(* POU with components common to all METS systems *)
PROGRAM C01_System
VAR
	fbCloseTCPSockets			: FB_SocketCloseAll;
	fbBasePath				: FB_SYSTEM_HardwareOS;
	//fbSystemFolders			: FB_SYSTEM_CreateFolders;
	fbCoreFolders			: FB_SYSTEM_CoreFolders;
	fbCorePaths				: FB_SYSTEM_CorePaths;
	
	fbMETSAppPath				: FB_SYSTEM_HardwareOS;
	fbMETSLogsPath				: FB_SYSTEM_HardwareOS;
	fbMETSProcessPath			: FB_SYSTEM_HardwareOS;
	
	bMETSApp_OK				: BOOL;
	bMETSLogs_OK			: BOOL;	
	bMETSProcess_OK			: BOOL;

	fbNVDataCtrl				: FB_CX_NVData_NOVRAM;
	fbSettings					: FB_CX_NVData_XMLFile;
	fbValidateSettings			: FB_SYSTEM_ValidateSettings;
	
	
	


	fbPulseNetwork			: FB_PulseGenerator;
	fbNetworkInfo				: FB_CX_NetworkInfo;
	aDisplayInfo				: ARRAY[1..6, 1..2] OF STRING(23);

	fbCloseTCPPorts			: FB_TCP_CloseAllPorts;
	fbTCPServerInitOK			: RS;

	fbDateTime				: FB_SYSTEM_DateTime;
	fbShiftMonitor				: FB_SYSTEM_ShiftMonitor;
	fbProdMonitor				: FB_SYSTEM_ProdMonitor;

	bManualChange: BOOL;
	bManualClosePorts		: BOOL;
	aNovRAMSize				: ARRAY[0..10] OF UDINT;

	fbDelayShutdown			: TON; 			(*Time to abort shutdown*)
	fbShutDown				: NT_Shutdown;
	fbAbortShutdown			: NT_AbortShutdown;
	nShutdownDelay			: DWORD;		(*Shutdown delay time*)

END_VAR
VAR // added by the converter: edge detectors and wires of the graphical bodies
    _w1 : BOOL;
END_VAR

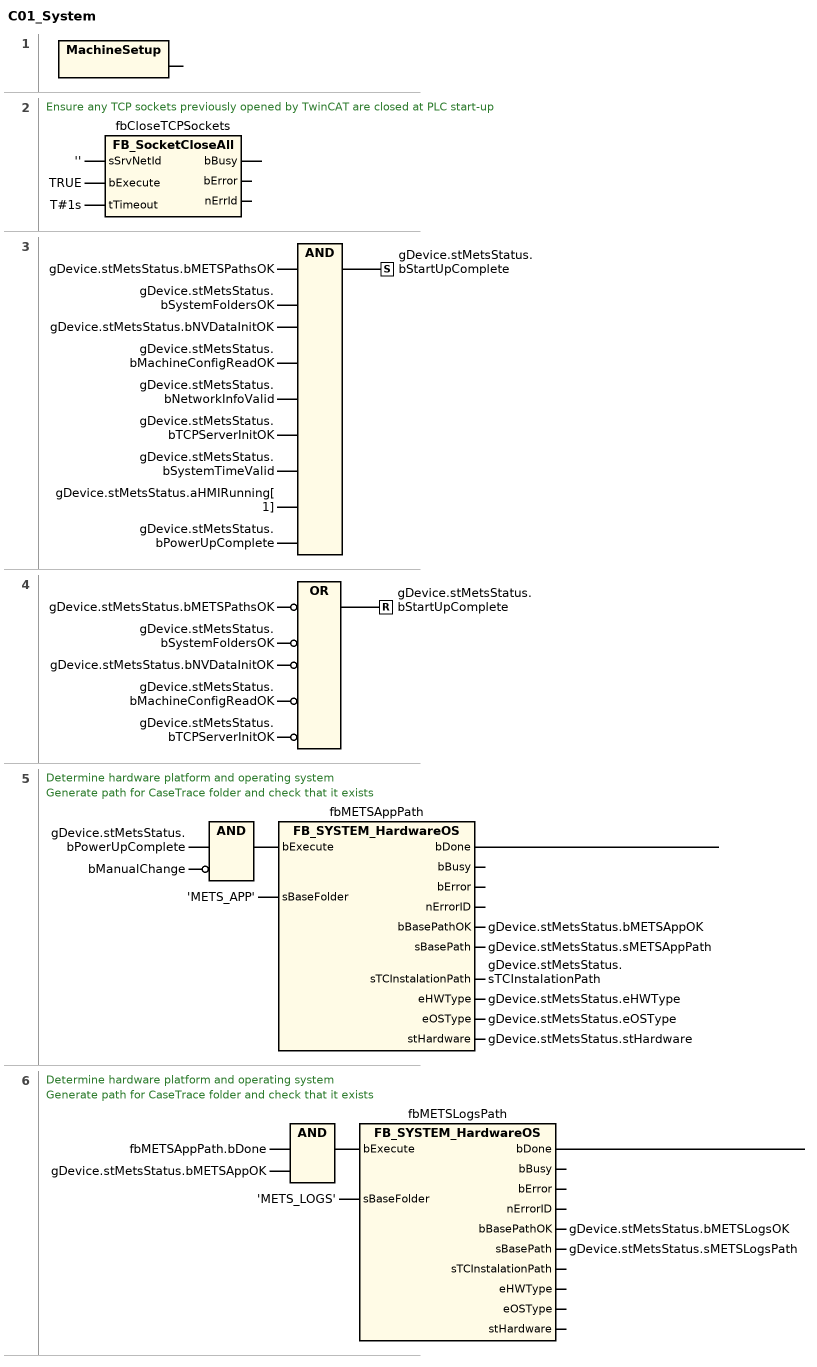
// NETWORK 1
MachineSetup();

// NETWORK 2
// Ensure any TCP sockets previously opened by TwinCAT are closed at PLC start-up
fbCloseTCPSockets(sSrvNetId := '', bExecute := TRUE, tTimeout := T#1s); // FB_SocketCloseAll

// NETWORK 3
gDevice.stMetsStatus.bStartUpComplete S= gDevice.stMetsStatus.bMETSPathsOK AND gDevice.stMetsStatus.bSystemFoldersOK AND gDevice.stMetsStatus.bNVDataInitOK AND gDevice.stMetsStatus.bMachineConfigReadOK AND gDevice.stMetsStatus.bNetworkInfoValid AND gDevice.stMetsStatus.bTCPServerInitOK AND gDevice.stMetsStatus.bSystemTimeValid AND gDevice.stMetsStatus.aHMIRunning[1] AND gDevice.stMetsStatus.bPowerUpComplete;

// NETWORK 4
gDevice.stMetsStatus.bStartUpComplete R= NOT gDevice.stMetsStatus.bMETSPathsOK OR NOT gDevice.stMetsStatus.bSystemFoldersOK OR NOT gDevice.stMetsStatus.bNVDataInitOK OR NOT gDevice.stMetsStatus.bMachineConfigReadOK OR NOT gDevice.stMetsStatus.bTCPServerInitOK;

// NETWORK 5
// 					Determine hardware platform and operating system
// Generate path for CaseTrace folder and check that it exists
//
fbMETSAppPath(
    bExecute := gDevice.stMetsStatus.bPowerUpComplete AND NOT bManualChange,
    sBaseFolder := 'METS_APP',
    bBasePathOK => gDevice.stMetsStatus.bMETSAppOK,
    sBasePath => gDevice.stMetsStatus.sMETSAppPath,
    sTCInstalationPath => gDevice.stMetsStatus.sTCInstalationPath,
    eHWType => gDevice.stMetsStatus.eHWType,
    eOSType => gDevice.stMetsStatus.eOSType,
    stHardware => gDevice.stMetsStatus.stHardware); // FB_SYSTEM_HardwareOS

// NETWORK 6
// 					Determine hardware platform and operating system
// Generate path for CaseTrace folder and check that it exists
//
fbMETSLogsPath(
    bExecute := fbMETSAppPath.bDone AND gDevice.stMetsStatus.bMETSAppOK,
    sBaseFolder := 'METS_LOGS',
    bBasePathOK => gDevice.stMetsStatus.bMETSLogsOK,
    sBasePath => gDevice.stMetsStatus.sMETSLogsPath); // FB_SYSTEM_HardwareOS

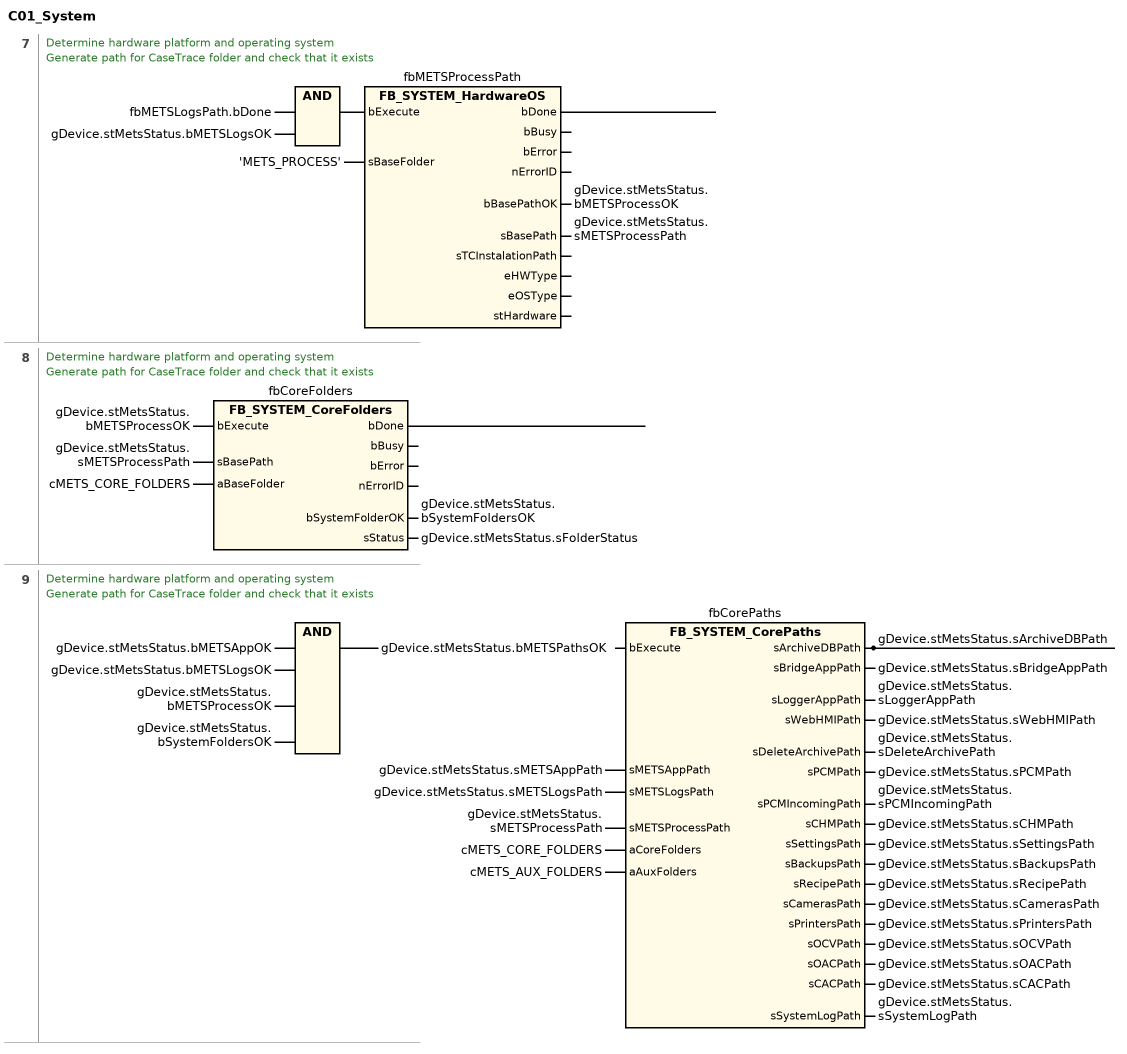
// NETWORK 7
// 					Determine hardware platform and operating system
// Generate path for CaseTrace folder and check that it exists
//
fbMETSProcessPath(
    bExecute := fbMETSLogsPath.bDone AND gDevice.stMetsStatus.bMETSLogsOK,
    sBaseFolder := 'METS_PROCESS',
    bBasePathOK => gDevice.stMetsStatus.bMETSProcessOK,
    sBasePath => gDevice.stMetsStatus.sMETSProcessPath); // FB_SYSTEM_HardwareOS

// NETWORK 8
// 					Determine hardware platform and operating system
// Generate path for CaseTrace folder and check that it exists
//
fbCoreFolders(
    bExecute := gDevice.stMetsStatus.bMETSProcessOK,
    sBasePath := gDevice.stMetsStatus.sMETSProcessPath,
    aBaseFolder := cMETS_CORE_FOLDERS,
    bSystemFolderOK => gDevice.stMetsStatus.bSystemFoldersOK,
    sStatus => gDevice.stMetsStatus.sFolderStatus); // FB_SYSTEM_CoreFolders

// NETWORK 9
// 					Determine hardware platform and operating system
// Generate path for CaseTrace folder and check that it exists
//
_w1 := gDevice.stMetsStatus.bMETSAppOK AND gDevice.stMetsStatus.bMETSLogsOK AND gDevice.stMetsStatus.bMETSProcessOK AND gDevice.stMetsStatus.bSystemFoldersOK;
gDevice.stMetsStatus.bMETSPathsOK := _w1;
fbCorePaths(
    bExecute := _w1,
    sMETSAppPath := gDevice.stMetsStatus.sMETSAppPath,
    sMETSLogsPath := gDevice.stMetsStatus.sMETSLogsPath,
    sMETSProcessPath := gDevice.stMetsStatus.sMETSProcessPath,
    aCoreFolders := cMETS_CORE_FOLDERS,
    aAuxFolders := cMETS_AUX_FOLDERS,
    sArchiveDBPath => gDevice.stMetsStatus.sArchiveDBPath,
    sBridgeAppPath => gDevice.stMetsStatus.sBridgeAppPath,
    sLoggerAppPath => gDevice.stMetsStatus.sLoggerAppPath,
    sWebHMIPath => gDevice.stMetsStatus.sWebHMIPath,
    sDeleteArchivePath => gDevice.stMetsStatus.sDeleteArchivePath,
    sPCMPath => gDevice.stMetsStatus.sPCMPath,
    sPCMIncomingPath => gDevice.stMetsStatus.sPCMIncomingPath,
    sCHMPath => gDevice.stMetsStatus.sCHMPath,
    sSettingsPath => gDevice.stMetsStatus.sSettingsPath,
    sBackupsPath => gDevice.stMetsStatus.sBackupsPath,
    sRecipePath => gDevice.stMetsStatus.sRecipePath,
    sCamerasPath => gDevice.stMetsStatus.sCamerasPath,
    sPrintersPath => gDevice.stMetsStatus.sPrintersPath,
    sOCVPath => gDevice.stMetsStatus.sOCVPath,
    sOACPath => gDevice.stMetsStatus.sOACPath,
    sCACPath => gDevice.stMetsStatus.sCACPath,
    sSystemLogPath => gDevice.stMetsStatus.sSystemLogPath); // FB_SYSTEM_CorePaths

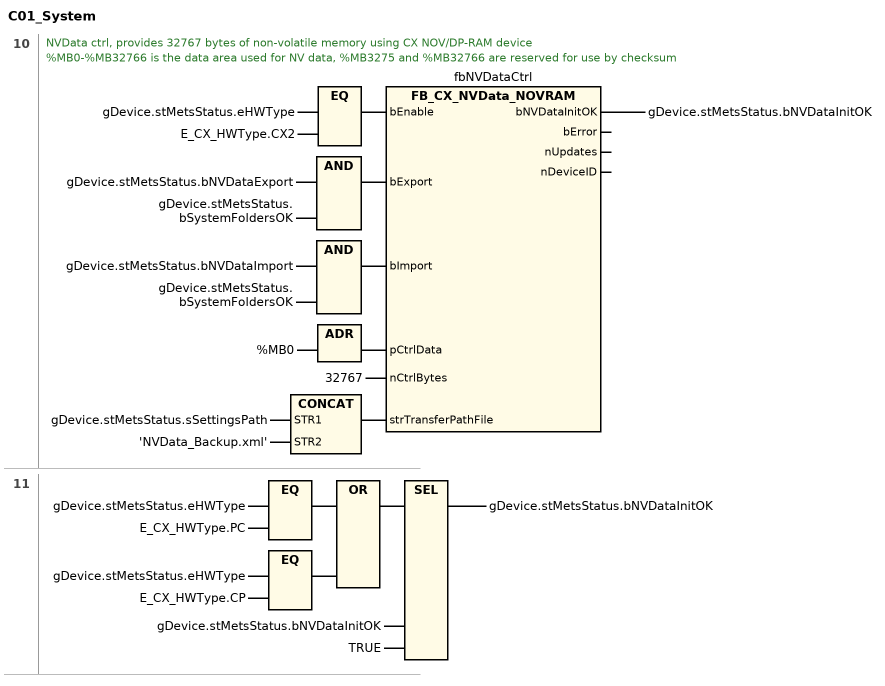
// NETWORK 10
// 					NVData ctrl, provides 32767 bytes of non-volatile memory using CX NOV/DP-RAM device
// %MB0-%MB32766 is the data area used for NV data, %MB3275 and %MB32766 are reserved for use by checksum
//
//
fbNVDataCtrl(
    bEnable := gDevice.stMetsStatus.eHWType = E_CX_HWType.CX2,
    bExport := gDevice.stMetsStatus.bNVDataExport AND gDevice.stMetsStatus.bSystemFoldersOK,
    bImport := gDevice.stMetsStatus.bNVDataImport AND gDevice.stMetsStatus.bSystemFoldersOK,
    pCtrlData := ADR(%MB0),
    nCtrlBytes := 32767,
    strTransferPathFile := CONCAT(STR1 := gDevice.stMetsStatus.sSettingsPath, STR2 := 'NVData_Backup.xml')); // FB_CX_NVData_NOVRAM
gDevice.stMetsStatus.bNVDataInitOK := fbNVDataCtrl.bNVDataInitOK;

// NETWORK 11
gDevice.stMetsStatus.bNVDataInitOK := SEL(gDevice.stMetsStatus.eHWType = E_CX_HWType.PC OR gDevice.stMetsStatus.eHWType = E_CX_HWType.CP, gDevice.stMetsStatus.bNVDataInitOK, TRUE);

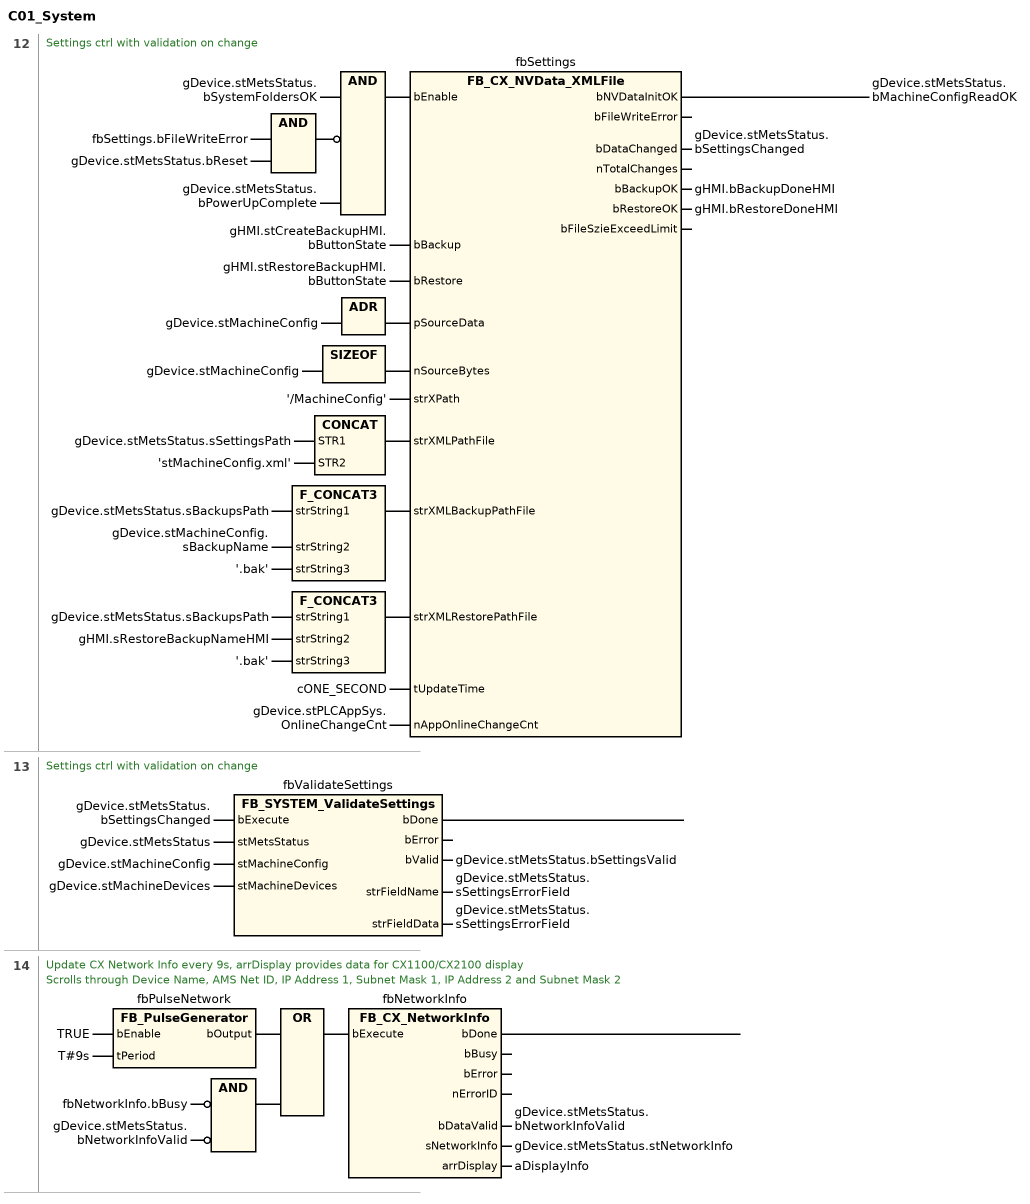
// NETWORK 12
// Settings ctrl with validation on change
fbSettings(
    bEnable := gDevice.stMetsStatus.bSystemFoldersOK AND NOT (fbSettings.bFileWriteError AND gDevice.stMetsStatus.bReset) AND gDevice.stMetsStatus.bPowerUpComplete,
    bBackup := gHMI.stCreateBackupHMI.bButtonState,
    bRestore := gHMI.stRestoreBackupHMI.bButtonState,
    pSourceData := ADR(gDevice.stMachineConfig),
    nSourceBytes := SIZEOF(gDevice.stMachineConfig),
    strXPath := '/MachineConfig',
    strXMLPathFile := CONCAT(STR1 := gDevice.stMetsStatus.sSettingsPath, STR2 := 'stMachineConfig.xml'),
    strXMLBackupPathFile := F_CONCAT3(strString1 := gDevice.stMetsStatus.sBackupsPath, strString2 := gDevice.stMachineConfig.sBackupName, strString3 := '.bak'),
    strXMLRestorePathFile := F_CONCAT3(strString1 := gDevice.stMetsStatus.sBackupsPath, strString2 := gHMI.sRestoreBackupNameHMI, strString3 := '.bak'),
    tUpdateTime := cONE_SECOND,
    nAppOnlineChangeCnt := gDevice.stPLCAppSys.OnlineChangeCnt,
    bDataChanged => gDevice.stMetsStatus.bSettingsChanged,
    bBackupOK => gHMI.bBackupDoneHMI,
    bRestoreOK => gHMI.bRestoreDoneHMI); // FB_CX_NVData_XMLFile
gDevice.stMetsStatus.bMachineConfigReadOK := fbSettings.bNVDataInitOK;

// NETWORK 13
// Settings ctrl with validation on change
fbValidateSettings(
    bExecute := gDevice.stMetsStatus.bSettingsChanged,
    stMetsStatus := gDevice.stMetsStatus,
    stMachineConfig := gDevice.stMachineConfig,
    stMachineDevices := gDevice.stMachineDevices,
    bValid => gDevice.stMetsStatus.bSettingsValid,
    strFieldName => gDevice.stMetsStatus.sSettingsErrorField,
    strFieldData => gDevice.stMetsStatus.sSettingsErrorField); // FB_SYSTEM_ValidateSettings

// NETWORK 14
// 					Update CX Network Info every 9s, arrDisplay provides data for CX1100/CX2100 display
// Scrolls through Device Name, AMS Net ID, IP Address 1, Subnet Mask 1, IP Address 2 and Subnet Mask 2
//
fbPulseNetwork(bEnable := TRUE, tPeriod := T#9s); // FB_PulseGenerator
fbNetworkInfo(
    bExecute := fbPulseNetwork.bOutput OR NOT fbNetworkInfo.bBusy AND NOT gDevice.stMetsStatus.bNetworkInfoValid,
    bDataValid => gDevice.stMetsStatus.bNetworkInfoValid,
    sNetworkInfo => gDevice.stMetsStatus.stNetworkInfo,
    arrDisplay => aDisplayInfo); // FB_CX_NetworkInfo

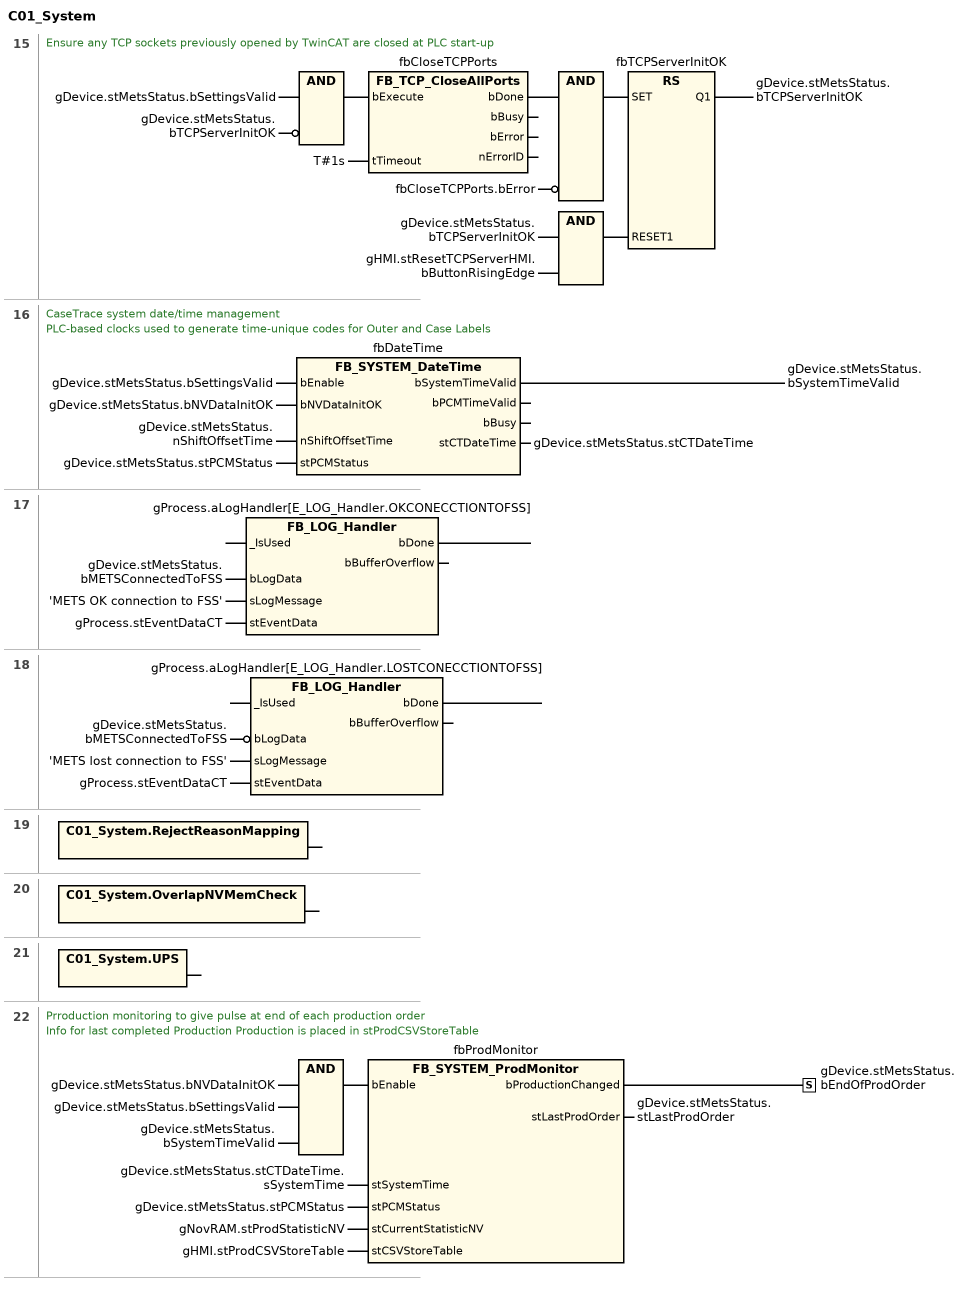
// NETWORK 15
// Ensure any TCP sockets previously opened by TwinCAT are closed at PLC start-up
fbCloseTCPPorts(bExecute := gDevice.stMetsStatus.bSettingsValid AND NOT gDevice.stMetsStatus.bTCPServerInitOK, tTimeout := T#1s); // FB_TCP_CloseAllPorts
fbTCPServerInitOK(SET := fbCloseTCPPorts.bDone AND NOT fbCloseTCPPorts.bError, RESET1 := gDevice.stMetsStatus.bTCPServerInitOK AND gHMI.stResetTCPServerHMI.bButtonRisingEdge); // RS
gDevice.stMetsStatus.bTCPServerInitOK := fbTCPServerInitOK.Q1;

// NETWORK 16
// 					CaseTrace system date/time management
// PLC-based clocks used to generate time-unique codes for Outer and Case Labels
//
fbDateTime(
    bEnable := gDevice.stMetsStatus.bSettingsValid,
    bNVDataInitOK := gDevice.stMetsStatus.bNVDataInitOK,
    nShiftOffsetTime := gDevice.stMetsStatus.nShiftOffsetTime,
    stPCMStatus := gDevice.stMetsStatus.stPCMStatus,
    stCTDateTime => gDevice.stMetsStatus.stCTDateTime); // FB_SYSTEM_DateTime
gDevice.stMetsStatus.bSystemTimeValid := fbDateTime.bSystemTimeValid;

// NETWORK 17
gProcess.aLogHandler[E_LOG_Handler.OKCONECCTIONTOFSS](
    bLogData := gDevice.stMetsStatus.bMETSConnectedToFSS,
    sLogMessage := 'METS OK connection to FSS',
    stEventData := gProcess.stEventDataCT); // FB_LOG_Handler

// NETWORK 18
gProcess.aLogHandler[E_LOG_Handler.LOSTCONECCTIONTOFSS](
    bLogData := NOT gDevice.stMetsStatus.bMETSConnectedToFSS,
    sLogMessage := 'METS lost connection to FSS',
    stEventData := gProcess.stEventDataCT); // FB_LOG_Handler

// NETWORK 19
C01_System.RejectReasonMapping();

// NETWORK 20
C01_System.OverlapNVMemCheck();

// NETWORK 21
C01_System.UPS();

// NETWORK 22
// 					Prroduction monitoring to give pulse at end of each production order
// Info for last completed Production Production is placed in stProdCSVStoreTable
//
fbProdMonitor(
    bEnable := gDevice.stMetsStatus.bNVDataInitOK AND gDevice.stMetsStatus.bSettingsValid AND gDevice.stMetsStatus.bSystemTimeValid,
    stSystemTime := gDevice.stMetsStatus.stCTDateTime.sSystemTime,
    stPCMStatus := gDevice.stMetsStatus.stPCMStatus,
    stCurrentStatisticNV := gNovRAM.stProdStatisticNV,
    stCSVStoreTable := gHMI.stProdCSVStoreTable,
    stLastProdOrder => gDevice.stMetsStatus.stLastProdOrder); // FB_SYSTEM_ProdMonitor
gDevice.stMetsStatus.bEndOfProdOrder S= fbProdMonitor.bProductionChanged;

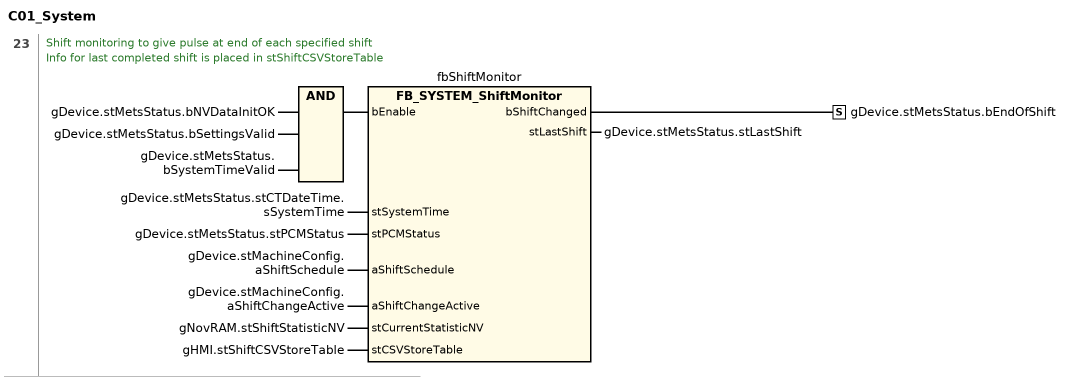
// NETWORK 23
// 					Shift monitoring to give pulse at end of each specified shift
// Info for last completed shift is placed in stShiftCSVStoreTable
//
fbShiftMonitor(
    bEnable := gDevice.stMetsStatus.bNVDataInitOK AND gDevice.stMetsStatus.bSettingsValid AND gDevice.stMetsStatus.bSystemTimeValid,
    stSystemTime := gDevice.stMetsStatus.stCTDateTime.sSystemTime,
    stPCMStatus := gDevice.stMetsStatus.stPCMStatus,
    aShiftSchedule := gDevice.stMachineConfig.aShiftSchedule,
    aShiftChangeActive := gDevice.stMachineConfig.aShiftChangeActive,
    stCurrentStatisticNV := gNovRAM.stShiftStatisticNV,
    stCSVStoreTable := gHMI.stShiftCSVStoreTable,
    stLastShift => gDevice.stMetsStatus.stLastShift); // FB_SYSTEM_ShiftMonitor
gDevice.stMetsStatus.bEndOfShift S= fbShiftMonitor.bShiftChanged;

ACTION MachineSetup:
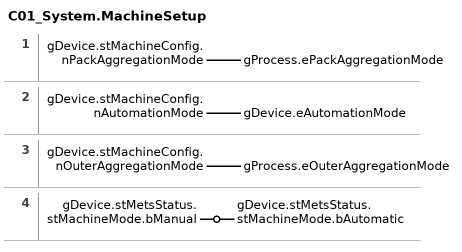
// NETWORK 1
gProcess.ePackAggregationMode := gDevice.stMachineConfig.nPackAggregationMode;

// NETWORK 2
gDevice.eAutomationMode := gDevice.stMachineConfig.nAutomationMode;

// NETWORK 3
gProcess.eOuterAggregationMode := gDevice.stMachineConfig.nOuterAggregationMode;

// NETWORK 4
gDevice.stMetsStatus.stMachineMode.bAutomatic := NOT gDevice.stMetsStatus.stMachineMode.bManual;
END_ACTION

ACTION OverlapNVMemCheck:
gMessage.nAlarm_OverlapNVMemCheck := 0;

IF ADR(gNovRAM.stMetsEfficiencyNV) -ADR( gNovRAM.stMetsCamerasNV) <= SIZEOF(gNovRAM.stMetsCamerasNV) THEN gMessage.nAlarm_OverlapNVMemCheck.0 := TRUE; END_IF
IF ADR(gNovRAM.stCasePackerSignalsNV) -ADR( gNovRAM.stMetsEfficiencyNV) <= SIZEOF(gNovRAM.stMetsEfficiencyNV) THEN gMessage.nAlarm_OverlapNVMemCheck.1 := TRUE; END_IF
IF ADR(gNovRAM.stCaseInspactionLogNV) -ADR( gNovRAM.stCasePackerSignalsNV) <= SIZEOF(gNovRAM.stCasePackerSignalsNV) THEN gMessage.nAlarm_OverlapNVMemCheck.2 := TRUE; END_IF
IF ADR(gNovRAM.sCurrentCHMArchiveDateNameNV) -ADR( gNovRAM.stCaseInspactionLogNV) <= SIZEOF(gNovRAM.stCaseInspactionLogNV) THEN gMessage.nAlarm_OverlapNVMemCheck.3 := TRUE; END_IF
IF ADR(gNovRAM.sNewCHMArchiveDateNameNV) -ADR( gNovRAM.sCurrentCHMArchiveDateNameNV) <= SIZEOF(gNovRAM.sCurrentCHMArchiveDateNameNV) THEN gMessage.nAlarm_OverlapNVMemCheck.4 := TRUE; END_IF
IF ADR(gNovRAM.sLastSendingTimeToFactoryLayerNV) -ADR( gNovRAM.sNewCHMArchiveDateNameNV) <= SIZEOF(gNovRAM.sNewCHMArchiveDateNameNV) THEN gMessage.nAlarm_OverlapNVMemCheck.5 := TRUE; END_IF
IF ADR(gNovRAM.stShiftStatisticNV) -ADR( gNovRAM.sLastSendingTimeToFactoryLayerNV) <= SIZEOF(gNovRAM.sLastSendingTimeToFactoryLayerNV) THEN gMessage.nAlarm_OverlapNVMemCheck.6 := TRUE; END_IF
IF ADR(gNovRAM.stProdStatisticNV) -ADR( gNovRAM.stShiftStatisticNV) <= SIZEOF(gNovRAM.stShiftStatisticNV) THEN gMessage.nAlarm_OverlapNVMemCheck.7 := TRUE; END_IF
IF ADR(gNovRAM.nNVChecksum) -ADR( gNovRAM.stProdStatisticNV) <= SIZEOF(gNovRAM.stProdStatisticNV) THEN gMessage.nAlarm_OverlapNVMemCheck.8 := TRUE; END_IF


(*Alarm bits list just to display status in conviniece view*)
gMessage.nAlarm_OverlapBitDisplay.1 := gMessage.nAlarm_OverlapNVMemCheck.1;
gMessage.nAlarm_OverlapBitDisplay.2 := gMessage.nAlarm_OverlapNVMemCheck.2;
gMessage.nAlarm_OverlapBitDisplay.3 := gMessage.nAlarm_OverlapNVMemCheck.3;
gMessage.nAlarm_OverlapBitDisplay.4 := gMessage.nAlarm_OverlapNVMemCheck.4;
gMessage.nAlarm_OverlapBitDisplay.5 := gMessage.nAlarm_OverlapNVMemCheck.5;
gMessage.nAlarm_OverlapBitDisplay.6 := gMessage.nAlarm_OverlapNVMemCheck.6;
gMessage.nAlarm_OverlapBitDisplay.7 := gMessage.nAlarm_OverlapNVMemCheck.7;
gMessage.nAlarm_OverlapBitDisplay.8 := gMessage.nAlarm_OverlapNVMemCheck.8;


aNovRAMSize[0] 	:= SIZEOF(gNovRAM.bInitBit);
aNovRAMSize[1]	:= SIZEOF(gNovRAM.stMetsCamerasNV);
aNovRAMSize[2] 	:= SIZEOF(gNovRAM.stMetsEfficiencyNV);
aNovRAMSize[3] 	:= SIZEOF(gNovRAM.stCasePackerSignalsNV);
aNovRAMSize[4] 	:= SIZEOF(gNovRAM.stCaseInspactionLogNV);
aNovRAMSize[5] 	:= SIZEOF(gNovRAM.sCurrentCHMArchiveDateNameNV);
aNovRAMSize[6] 	:= SIZEOF(gNovRAM.sNewCHMArchiveDateNameNV);
aNovRAMSize[7] 	:= SIZEOF(gNovRAM.sLastSendingTimeToFactoryLayerNV);
aNovRAMSize[8] 	:= SIZEOF(gNovRAM.stShiftStatisticNV);
aNovRAMSize[9]	:= SIZEOF(gNovRAM.stProdStatisticNV);
aNovRAMSize[10]	:= SIZEOF(gNovRAM.nNVChecksum);
END_ACTION

ACTION RejectReasonMapping:
(*********************Reject Code Mapping for Shift Statistic****************************)

 gProcess.aRejectCountersID[0] := gProcess.stPackRejectReasons.stUnknownPackReject.nRejectID;  (*'UnknownReason';*)
 gProcess.aRejectCountersID[1] := gProcess.stPackRejectReasons.stPackCodesNotLinked.nRejectID; (*'Pack code(s) not linked';*)
 gProcess.aRejectCountersID[2] := gProcess.stPackRejectReasons.stPackCodesOverwritten.nRejectID; (* 'Pack code(s) over-written';*)
 gProcess.aRejectCountersID[3] := gProcess.stPackRejectReasons.stPackCodesGtinError.nRejectID; (* 'Pack code(s) invalid GTIN';*)
 gProcess.aRejectCountersID[4] := gProcess.stPackRejectReasons.stPackCodesSerialError.nRejectID; (*'Pack code(s) invalid Serial Code';*)
 gProcess.aRejectCountersID[5] := gProcess.stPackRejectReasons.stPackCodeInvalidLength.nRejectID; (*'Pack code(s) invalid Length';*)
 gProcess.aRejectCountersID[6] := gProcess.stPackRejectReasons.stPackCodesNotRead.nRejectID; (*'Pack code(s) no read';*)
 gProcess.aRejectCountersID[7] := gProcess.stPackRejectReasons.stPackCodesDuplicated.nRejectID; (*'Pack code(s) duplicate';*)
 gProcess.aRejectCountersID[8] := gProcess.stPackRejectReasons.stPackCodesTypeError.nRejectID; (*'Pack code(s) invalid type';*)
 gProcess.aRejectCountersID[9] := gProcess.stPackRejectReasons.stPackCodesSUPIError.nRejectID; (*'Pack code(s) SUPI failed validation';*)
 gProcess.aRejectCountersID[10] := gProcess.stPackRejectReasons.stPackCodesDBError.nRejectID;  (*'Pack code DB failed validation';*)
 gProcess.aRejectCountersID[11] := gProcess.stPackRejectReasons.stPackCodesBrandSpec.nRejectID; (*'Pack code(s) invalid Brand';*)
 gProcess.aRejectCountersID[12] := 1000;
 gProcess.aRejectCountersID[13] := 1000;
 gProcess.aRejectCountersID[14] := 1000;
 gProcess.aRejectCountersID[15] := 1000;
 gProcess.aRejectCountersID[16] := 1000;
 gProcess.aRejectCountersID[17] := 1000;
 gProcess.aRejectCountersID[18] := 1000;
 gProcess.aRejectCountersID[19] := 1000;

 gProcess.aRejectCountersID[20] := gProcess.stOuterRejectReasons.stUnknownOuterReject.nRejectID;  (*'UnknownReason';*)
 gProcess.aRejectCountersID[21] := gProcess.stOuterRejectReasons.stOuterBarcodeGtinError.nRejectID; (*'GTIN';*)
 gProcess.aRejectCountersID[22] := gProcess.stOuterRejectReasons.stOuterBarcodeRskuError.nRejectID; (*'RSKU';*)
 gProcess.aRejectCountersID[23] := gProcess.stOuterRejectReasons.stOuterCodeSerialError.nRejectID; (*'Serial';*)
 gProcess.aRejectCountersID[24] := gProcess.stOuterRejectReasons.stOuterBarcodeInvalidLength.nRejectID; (*'Length';*)
 gProcess.aRejectCountersID[25] := gProcess.stOuterRejectReasons.stOuterBarcodeNotRead.nRejectID; (*'Outer code Not Read';*)
 gProcess.aRejectCountersID[26] := gProcess.stOuterRejectReasons.stOuterBarcodeDuplicate.nRejectID; (*'code duplicate';*)
 gProcess.aRejectCountersID[27] := gProcess.stOuterRejectReasons.stOuterDataNotFound.nRejectID; (* '(OAC) not found ';*)
 gProcess.aRejectCountersID[28] := gProcess.stOuterRejectReasons.stOuterGeneralCodeError.nRejectID; (* 'Outer Label not read';*)
 gProcess.aRejectCountersID[29] := gProcess.stOuterRejectReasons.stOuterTimeOutValidation.nRejectID; (* 'Validation Timeout';*)
 gProcess.aRejectCountersID[30] := gProcess.stOuterRejectReasons.stOuterDuplicatedPackCodesFound.nRejectID; (*'duplicate pack codes';*)
 gProcess.aRejectCountersID[31] := gProcess.stOuterRejectReasons.stOuterPackCodeDataNotFound.nRejectID; (*'OCV';*)
 gProcess.aRejectCountersID[32] := gProcess.stOuterRejectReasons.stOuterConfirmCodeNotRead.nRejectID; (*'confirmation pack code(s)';*)
 gProcess.aRejectCountersID[33] := gProcess.stOuterRejectReasons.stOuterPackCodeNotRead.nRejectID; (*'acceptance level';*)
 gProcess.aRejectCountersID[34] := gProcess.stOuterRejectReasons.stOuterPackCodeInvalid.nRejectID; (*'QA';*)
 gProcess.aRejectCountersID[35] := gProcess.stOuterRejectReasons.stOuterQAReject.nRejectID; (*'QA';*)
 gProcess.aRejectCountersID[36] := gProcess.stOuterRejectReasons.stOuterPackCodeDBError.nRejectID; (*'pack codes DB Error';*)
 gProcess.aRejectCountersID[37] := gProcess.stOuterRejectReasons.stOuterBarcodeDBError.nRejectID; (*'Outer code DB Error';*)
 gProcess.aRejectCountersID[38] := gProcess.stOuterRejectReasons.stOuterCodesBrandSpecError.nRejectID; (*'Outer code invalid Brand'*)
 gProcess.aRejectCountersID[39] := 1000;
 gProcess.aRejectCountersID[40] := 1000;
 gProcess.aRejectCountersID[41] := 1000;
 gProcess.aRejectCountersID[42] := 1000;
 gProcess.aRejectCountersID[43] := 1000;
 gProcess.aRejectCountersID[44] := 1000;
 gProcess.aRejectCountersID[45] := 1000;
 gProcess.aRejectCountersID[46] := 1000;
 gProcess.aRejectCountersID[47] := 1000;
 gProcess.aRejectCountersID[48] := 1000;
 gProcess.aRejectCountersID[49] := 1000;

 gProcess.aRejectCountersID[50] := gProcess.stCaseRejectReasons.stUnknownCaseReject.nRejectID;  (*'UnknownReason';*)
 gProcess.aRejectCountersID[51] := gProcess.stCaseRejectReasons.stValError.nRejectID; (*'VAL';*)		(*cINIT_CASE_REJECT_INDEX*)
 gProcess.aRejectCountersID[52] := gProcess.stCaseRejectReasons.stOACError.nRejectID; (*'OAC';*)
 gProcess.aRejectCountersID[53] := gProcess.stCaseRejectReasons.stINVError.nRejectID; (*'INV';*)
 gProcess.aRejectCountersID[54] := gProcess.stCaseRejectReasons.stDUPError.nRejectID; (*'DUP';*)
 gProcess.aRejectCountersID[55] := gProcess.stCaseRejectReasons.stPackNotLinedError.nRejectID; (*'PACK';*)
 gProcess.aRejectCountersID[56] := gProcess.stCaseRejectReasons.stOuterGTINError.nRejectID; (*'OUTERGTIN';*)
 gProcess.aRejectCountersID[57] := gProcess.stCaseRejectReasons.stOuterSerialError.nRejectID; (*'OUTERSER';*)
 gProcess.aRejectCountersID[58] := gProcess.stCaseRejectReasons.stOuterRSKUError.nRejectID; (* 'OUTERSKU';*)
 gProcess.aRejectCountersID[59] := gProcess.stCaseRejectReasons.stNoCaseLabelError.nRejectID; (*'NOCASELABEL';*)
 gProcess.aRejectCountersID[60] := gProcess.stCaseRejectReasons.stCasePackerReject.nRejectID; (*'CASEPACKERREJECT';*)
 gProcess.aRejectCountersID[61] := gProcess.stCaseRejectReasons.stDoorGuardReject.nRejectID; (*'DOORGUARDREJECT';*)
 gProcess.aRejectCountersID[62] := gProcess.stCaseRejectReasons.stCaseLabelGtinError.nRejectID; (*'CASEGTIN';*)
 gProcess.aRejectCountersID[63] := gProcess.stCaseRejectReasons.stCaseLabelRskuError.nRejectID;(*'CASESKU';*)
 gProcess.aRejectCountersID[64] := gProcess.stCaseRejectReasons.stCaseLabelProductionOrderError.nRejectID; (*'CASEPROD';*)
 gProcess.aRejectCountersID[65] := gProcess.stCaseRejectReasons.stCaseLabelBatchIDError.nRejectID; (*'CASEBATCHID';*)
 gProcess.aRejectCountersID[66] := gProcess.stCaseRejectReasons.stCaseLabelSerialCodeError.nRejectID; (*'CASESERIALCODE';*)
 gProcess.aRejectCountersID[67] := gProcess.stCaseRejectReasons.stCaseLabelDuplicate.nRejectID; (*'DUPCASELABEL';*)
 gProcess.aRejectCountersID[68] := gProcess.stCaseRejectReasons.stCaseNoCaseData.nRejectID; (*'NOCASEDATA';*)
 gProcess.aRejectCountersID[69] := gProcess.stCaseRejectReasons.stCaseBarcodeInvalidLength.nRejectID; (*'CASECODELENGTH';*)
 gProcess.aRejectCountersID[70] := gProcess.stCaseRejectReasons.stCaseDBInvalidCheck.nRejectID; (*'CACDBINVALID';*)
 gProcess.aRejectCountersID[71] := gProcess.stCaseRejectReasons.stCaseWhitelistInvalidCheck.nRejectID; (*'OHMWHITELIST';*)
 gProcess.aRejectCountersID[72] := gProcess.stCaseRejectReasons.stOuterBrandError.nRejectID; (*OUTERSBRAND*)
 gProcess.aRejectCountersID[73] := gProcess.stCaseRejectReasons.stCaseLabelBrandCodeError.nRejectID; (*CASEBRAND*)
 gProcess.aRejectCountersID[74] := 1000;
 gProcess.aRejectCountersID[75] := 1000;
 gProcess.aRejectCountersID[76] := 1000;
 gProcess.aRejectCountersID[77] := 1000;
 gProcess.aRejectCountersID[78] := 1000;
 gProcess.aRejectCountersID[79] := 1000;
 gProcess.aRejectCountersID[80] := 1000;
END_ACTION

ACTION UPS:
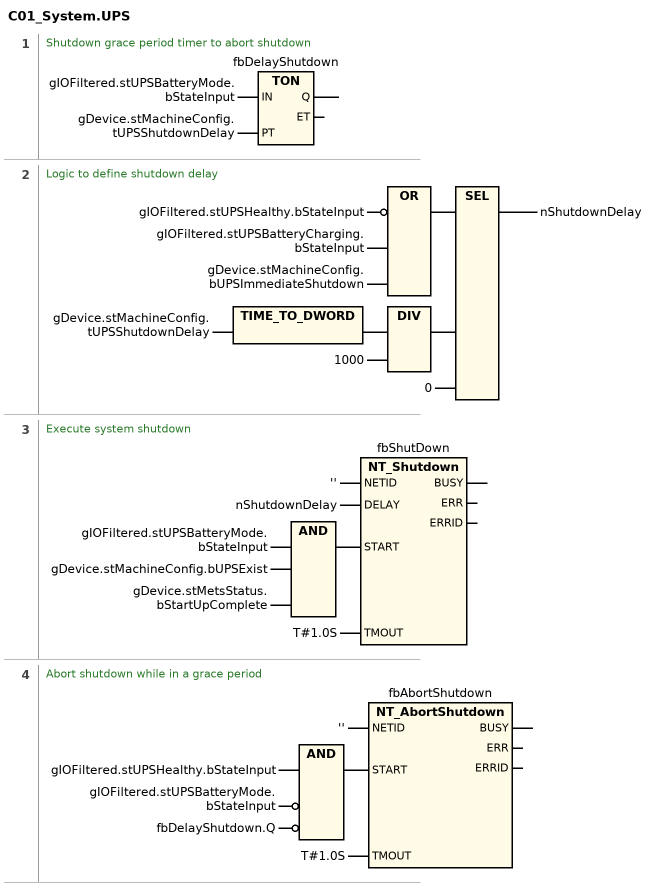
// NETWORK 1
// Shutdown grace period timer to abort shutdown
fbDelayShutdown(IN := gIOFiltered.stUPSBatteryMode.bStateInput, PT := gDevice.stMachineConfig.tUPSShutdownDelay); // TON

// NETWORK 2
// Logic to define shutdown delay
nShutdownDelay := SEL(NOT gIOFiltered.stUPSHealthy.bStateInput OR gIOFiltered.stUPSBatteryCharging.bStateInput OR gDevice.stMachineConfig.bUPSImmediateShutdown, TIME_TO_DWORD(gDevice.stMachineConfig.tUPSShutdownDelay) / 1000, 0);

// NETWORK 3
// Execute system shutdown
fbShutDown(
    NETID := '',
    DELAY := nShutdownDelay,
    START := gIOFiltered.stUPSBatteryMode.bStateInput AND gDevice.stMachineConfig.bUPSExist AND gDevice.stMetsStatus.bStartUpComplete,
    TMOUT := T#1.0S); // NT_Shutdown

// NETWORK 4
// Abort shutdown while in a grace period
fbAbortShutdown(
    NETID := '',
    START := gIOFiltered.stUPSHealthy.bStateInput AND NOT gIOFiltered.stUPSBatteryMode.bStateInput AND NOT fbDelayShutdown.Q,
    TMOUT := T#1.0S); // NT_AbortShutdown
END_ACTION

END_PROGRAM

(* stored: Version 1.1.0.1
   POU C01_System: Id {05763847-fc71-4ec4-95d0-dda019cef70f}, SpecialFunc None
   Action MachineSetup: Id {edc125aa-7185-4f61-8a35-fcbc5b05e805}
   Action OverlapNVMemCheck: Id {2db2671e-b517-4d81-9841-2ae9aec1008e}
   Action RejectReasonMapping: Id {d5b2d0b7-242b-4ef2-a1d8-0fd66bd57188}
   Action UPS: Id {f8b3f222-aba0-4a75-92fe-946159efc17b} *)
